(* PLC project Aufgabenserie_3, Beckhoff Automation GmbH TwinCAT PLC Control 3.5.10.30 *)
(* stored: creationDateTime 2018-11-15T20:00:53.5125784, modificationDateTime 2018-11-15T20:00:53.5156126 *)

FUNCTION_BLOCK fb_edgeDetector
VAR_INPUT
	b_inputVal			:	BOOL;
	i_doobleActivTime	: 	INT			:=50;
END_VAR
VAR_OUTPUT
	b_risingEdge		:	BOOL;
	b_doubleActivate	:	BOOL;
	b_fallingEdge		:	BOOL;
END_VAR
VAR
	b_state				:	BOOL;
	i_timCnt			:	INT;
	i_debCnt			:	INT		:=0;
	
	st_current_state		:	FSM_Deb	:= FSM_Deb.deb_state_init;
END_VAR

            b_risingEdge		:= 	FALSE;
b_fallingEdge		:=	FALSE;
b_doubleActivate	:=	FALSE;
CASE st_current_state OF
	FSM_Deb.deb_state_init:
		IF b_inputVal THEN
			st_current_state	:=	FSM_Deb.deb_state_high;
		ELSE
			st_current_state	:=	FSM_Deb.deb_state_low;
		END_IF
	
	FSM_Deb.deb_state_low:
		IF b_inputVal THEN
			st_current_state	:=	FSM_Deb.deb_state_rising;
		END_IF
		
	FSM_Deb.deb_state_rising:
		IF i_debCnt<5 THEN
			i_debCnt	:= i_debCnt+1;
		ELSIF i_debCnt<i_doobleActivTime THEN
			i_debCnt	:= i_debCnt+1;
			IF NOT b_inputVal THEN
				st_current_state	:=	FSM_Deb.deb_state_doble_activ;
			END_IF
		ELSE
			b_risingEdge			:= TRUE;
			st_current_state		:=	FSM_Deb.deb_state_high;
			i_debCnt				:= 0;
		END_IF
	
	FSM_Deb.deb_state_doble_activ:
		IF i_debCnt<i_doobleActivTime THEN
			IF b_inputVal THEN
				b_doubleActivate	:= TRUE;
				st_current_state	:=	FSM_Deb.deb_state_high;
				i_debCnt			:=0;
			ELSE
				i_debCnt		:= i_debCnt+1;
			END_IF
		ELSE
			st_current_state	:=	FSM_Deb.deb_state_low;
			i_debCnt			:=0;
			
		END_IF
	
	FSM_Deb.deb_state_high:
		IF NOT b_inputVal THEN
			st_current_state	:= FSM_Deb.deb_state_falling;
		END_IF
	
	FSM_Deb.deb_state_falling:
		IF i_debCnt<1 THEN
			i_debCnt	:= i_debCnt+1;
		ELSE
			st_current_state	:=	FSM_deb.deb_state_low;
			b_fallingEdge		:= TRUE;		
			i_debCnt			:=0;
		END_IF
	
		
END_CASE

          
END_FUNCTION_BLOCK
